LIN {X 0,Y 290.897,Z 639.692,A -85,B 0,C 180,E1 -29510.461,E2 -29510.461} C_VEL
LIN {X 0,Y 298.304,Z 601.913,A -85,B 0,C 180,E1 -29511.106,E2 -29511.106} C_VEL
LIN {X 0,Y 304.521,Z 561.656,A -85,B 0,C 180,E1 -29511.707,E2 -29511.707} C_VEL
LIN {X 0,Y 310.827,Z 508.179,A -85,B 0,C 180,E1 -29512.467,E2 -29512.467} C_VEL
LIN {X 0,Y 310.206,Z 504.294,A -85,B 0,C 180,E1 -29514.876,E2 -29514.876} C_VEL
LIN {X 0,Y 310.624,Z 502.045,A -85,B 0,C 180,E1 -29517.048,E2 -29517.048} C_VEL
LIN {X 0,Y 311.19,Z 500.451,A -85,B 0,C 180,E1 -29519.079,E2 -29519.079} C_VEL
LIN {X 0,Y 311.684,Z 500.279,A -85,B 0,C 180,E1 -29520.807,E2 -29520.807} C_VEL
LIN {X 0,Y 307.357,Z 520.155,A -85,B 0,C 180,E1 -29521.159,E2 -29521.159} C_VEL
LIN {X 0,Y 298.937,Z 587.892,A -85,B 0,C 180,E1 -29522.314,E2 -29522.314} C_VEL
LIN {X 0,Y 292.33,Z 627.482,A -85,B 0,C 180,E1 -29522.975,E2 -29522.975} C_VEL
LIN {X 0,Y 283.931,Z 667.082,A -85,B 0,C 180,E1 -29523.677,E2 -29523.677} C_VEL
LIN {X 0,Y 273.634,Z 706.852,A -85,B 0,C 180,E1 -29524.571,E2 -29524.571} C_VEL
LIN {X 0,Y 273.269,Z 708.115,A -85,B 0,C 180,E1 -29524.603,E2 -29524.603} C_VEL
LIN {X 0,Y 270.934,Z 715.53,A -85,B 0,C 180,E1 -29524.577,E2 -29524.577} C_VEL
LIN {X 0,Y 264.164,Z 735.315,A -85,B 0,C 180,E1 -29523.788,E2 -29523.788} C_VEL
LIN {X 0,Y 261.988,Z 741.59,A -85,B 0,C 180,E1 -29523.82,E2 -29523.82} C_VEL
LIN {X 0,Y 253.319,Z 766.281,A -85,B 0,C 180,E1 -29524.687,E2 -29524.687} C_VEL
LIN {X 0,Y 244.331,Z 786.818,A -85,B 0,C 180,E1 -29525.636,E2 -29525.636} C_VEL
LIN {X 0,Y 234.279,Z 805.781,A -85,B 0,C 180,E1 -29526.721,E2 -29526.721} C_VEL
LIN {X 0,Y 222.708,Z 824.293,A -85,B 0,C 180,E1 -29528.119,E2 -29528.119} C_VEL
LIN {X 0,Y 210.064,Z 841.669,A -85,B 0,C 180,E1 -29529.835,E2 -29529.835} C_VEL
LIN {X 0,Y 196.263,Z 858.133,A -85,B 0,C 180,E1 -29531.994,E2 -29531.994} C_VEL
LIN {X 0,Y 181.928,Z 873.186,A -85,B 0,C 180,E1 -29534.691,E2 -29534.691} C_VEL
LIN {X 0,Y 167.238,Z 886.889,A -85,B 0,C 180,E1 -29538.078,E2 -29538.078} C_VEL
LIN {X 0,Y 152.362,Z 899.309,A -85,B 0,C 180,E1 -29542.373,E2 -29542.373} C_VEL
LIN {X 0,Y 137.965,Z 910.277,A -85,B 0,C 180,E1 -29547.849,E2 -29547.849} C_VEL
LIN {X 0,Y 124.37,Z 919.877,A -85,B 0,C 180,E1 -29554.911,E2 -29554.911} C_VEL
LIN {X 0,Y 112.547,Z 927.982,A -85,B 0,C 180,E1 -29563.977,E2 -29563.977} C_VEL
LIN {X 0,Y 103.618,Z 934.442,A -85,B 0,C 180,E1 -29575.297,E2 -29575.297} C_VEL
LIN {X 0,Y 99.045,Z 938.841,A -85,B 0,C 180,E1 -29587.442,E2 -29587.442} C_VEL
LIN {X 0,Y 98.366,Z 941.455,A -85,B 0,C 180,E1 -29599.458,E2 -29599.458} C_VEL
LIN {X 0,Y 99.632,Z 942.357,A -85,B 0,C 180,E1 -29608.275,E2 -29608.275} C_VEL
LIN {X 0,Y 99.687,Z 942.359,A -85,B 0,C 180,E1 -29611.725,E2 -29611.725} C_VEL
LIN {X 0,Y 98.619,Z 941.398,A -85,B 0,C 180,E1 -29621.107,E2 -29621.107} C_VEL
LIN {X 0,Y 100.203,Z 938.422,A -85,B 0,C 180,E1 -29634.15,E2 -29634.15} C_VEL
LIN {X 0,Y 106.237,Z 933.564,A -85,B 0,C 180,E1 -29646.367,E2 -29646.367} C_VEL
LIN {X 0,Y 116.506,Z 926.832,A -85,B 0,C 180,E1 -29656.845,E2 -29656.845} C_VEL
LIN {X 0,Y 119.403,Z 925.309,A -85,B 0,C 180,E1 -29658.909,E2 -29658.909} C_VEL
LIN {X 0,Y 124.749,Z 925.094,A -85,B 0,C 180,E1 -29662.895,E2 -29662.895} C_VEL
LIN {X 0,Y 116.212,Z 919.228,A -85,B 0,C 180,E1 -29668.919,E2 -29668.919} C_VEL
LIN {X 0,Y 105.712,Z 915.062,A -85,B 0,C 180,E1 -29682.382,E2 -29682.382} C_VEL
LIN {X 0,Y 102.911,Z 908.863,A -85,B 0,C 180,E1 -29705.576,E2 -29705.576} C_VEL
LIN {X 0,Y 125.546,Z 900.271,A -85,B 0,C 180,E1 -29734.076,E2 -29734.076} C_VEL
LIN {X 0,Y 136.876,Z 897.562,A -85,B 0,C 180,E1 -29739.911,E2 -29739.911} C_VEL
LIN {X 0,Y 124.152,Z 904.891,A -85,B 0,C 180,E1 -29747.427,E2 -29747.427} C_VEL
LIN {X 0,Y 113.258,Z 910.617,A -85,B 0,C 180,E1 -29756.813,E2 -29756.813} C_VEL
LIN {X 0,Y 105.415,Z 914.504,A -85,B 0,C 180,E1 -29767.702,E2 -29767.702} C_VEL
LIN {X 0,Y 101.161,Z 916.605,A -85,B 0,C 180,E1 -29779.175,E2 -29779.175} C_VEL
LIN {X 0,Y 99.972,Z 917.237,A -85,B 0,C 180,E1 -29790.573,E2 -29790.573} C_VEL
LIN {X 0,Y 101.413,Z 916.524,A -85,B 0,C 180,E1 -29801.949,E2 -29801.949} C_VEL
LIN {X 0,Y 106.246,Z 914.18,A -85,B 0,C 180,E1 -29813.871,E2 -29813.871} C_VEL
LIN {X 0,Y 114.517,Z 910.086,A -85,B 0,C 180,E1 -29824.579,E2 -29824.579} C_VEL
LIN {X 0,Y 125.775,Z 904.102,A -85,B 0,C 180,E1 -29833.759,E2 -29833.759} C_VEL
LIN {X 0,Y 138.765,Z 896.517,A -85,B 0,C 180,E1 -29841.096,E2 -29841.096} C_VEL
LIN {X 0,Y 152.72,Z 887.421,A -85,B 0,C 180,E1 -29846.934,E2 -29846.934} C_VEL
LIN {X 0,Y 167.084,Z 876.867,A -85,B 0,C 180,E1 -29851.606,E2 -29851.606} C_VEL
LIN {X 0,Y 181.46,Z 864.89,A -85,B 0,C 180,E1 -29855.394,E2 -29855.394} C_VEL
LIN {X 0,Y 195.585,Z 851.485,A -85,B 0,C 180,E1 -29858.503,E2 -29858.503} C_VEL
LIN {X 0,Y 208.601,Z 837.38,A -85,B 0,C 180,E1 -29860.977,E2 -29860.977} C_VEL
LIN {X 0,Y 221.053,Z 821.901,A -85,B 0,C 180,E1 -29863.073,E2 -29863.073} C_VEL
LIN {X 0,Y 232.13,Z 806.011,A -85,B 0,C 180,E1 -29864.768,E2 -29864.768} C_VEL
LIN {X 0,Y 241.983,Z 789.593,A -85,B 0,C 180,E1 -29866.176,E2 -29866.176} C_VEL
LIN {X 0,Y 250.51,Z 772.939,A -85,B 0,C 180,E1 -29867.343,E2 -29867.343} C_VEL
LIN {X 0,Y 258.342,Z 754.518,A -85,B 0,C 180,E1 -29868.389,E2 -29868.389} C_VEL
LIN {X 0,Y 264.963,Z 735.092,A -85,B 0,C 180,E1 -29869.289,E2 -29869.289} C_VEL
LIN {X 0,Y 274.717,Z 701.51,A -85,B 0,C 180,E1 -29870.526,E2 -29870.526} C_VEL
LIN {X 0,Y 283.63,Z 667.686,A -85,B 0,C 180,E1 -29871.459,E2 -29871.459} C_VEL
LIN {X 0,Y 292.295,Z 629.172,A -85,B 0,C 180,E1 -29872.213,E2 -29872.213} C_VEL
LIN {X 0,Y 299.95,Z 586.992,A -85,B 0,C 180,E1 -29872.859,E2 -29872.859} C_VEL
LIN {X 0,Y 305.774,Z 544.445,A -85,B 0,C 180,E1 -29873.432,E2 -29873.432} C_VEL
LIN {X 0,Y 309.314,Z 514.061,A -85,B 0,C 180,E1 -29873.83,E2 -29873.83} C_VEL
LIN {X 0,Y 308.742,Z 510.419,A -85,B 0,C 180,E1 -29876.472,E2 -29876.472} C_VEL
LIN {X 0,Y 309.391,Z 508.21,A -85,B 0,C 180,E1 -29879.259,E2 -29879.259} C_VEL
LIN {X 0,Y 309.404,Z 508.336,A -85,B 0,C 180,E1 -29879.467,E2 -29879.467} C_VEL
LIN {X 0,Y 307.496,Z 517.679,A -85,B 0,C 180,E1 -29879.622,E2 -29879.622} C_VEL
LIN {X 0,Y 298.935,Z 585.198,A -85,B 0,C 180,E1 -29880.732,E2 -29880.732} C_VEL
LIN {X 0,Y 292.245,Z 624.865,A -85,B 0,C 180,E1 -29881.368,E2 -29881.368} C_VEL
LIN {X 0,Y 283.725,Z 664.756,A -85,B 0,C 180,E1 -29882.02,E2 -29882.02} C_VEL
LIN {X 0,Y 273.246,Z 704.978,A -85,B 0,C 180,E1 -29882.855,E2 -29882.855} C_VEL
LIN {X 0,Y 261.988,Z 741.59,A -85,B 0,C 180,E1 -29883.82,E2 -29883.82} C_VEL
LIN {X 0,Y 259.38,Z 748.91,A -85,B 0,C 180,E1 -29883.841,E2 -29883.841} C_VEL
LIN {X 0,Y 252.021,Z 767.378,A -85,B 0,C 180,E1 -29883.147,E2 -29883.147} C_VEL
LIN {X 0,Y 248.861,Z 774.441,A -85,B 0,C 180,E1 -29883.206,E2 -29883.206} C_VEL
LIN {X 0,Y 239.587,Z 793.606,A -85,B 0,C 180,E1 -29884.102,E2 -29884.102} C_VEL
LIN {X 0,Y 228.912,Z 812.088,A -85,B 0,C 180,E1 -29885.187,E2 -29885.187} C_VEL
LIN {X 0,Y 216.891,Z 829.847,A -85,B 0,C 180,E1 -29886.549,E2 -29886.549} C_VEL
LIN {X 0,Y 203.66,Z 846.745,A -85,B 0,C 180,E1 -29888.28,E2 -29888.28} C_VEL
LIN {X 0,Y 189.138,Z 862.871,A -85,B 0,C 180,E1 -29890.487,E2 -29890.487} C_VEL
LIN {X 0,Y 173.667,Z 877.908,A -85,B 0,C 180,E1 -29893.34,E2 -29893.34} C_VEL
LIN {X 0,Y 157.883,Z 891.47,A -85,B 0,C 180,E1 -29897.001,E2 -29897.001} C_VEL
LIN {X 0,Y 142.882,Z 902.971,A -85,B 0,C 180,E1 -29901.451,E2 -29901.451} C_VEL
LIN {X 0,Y 128.217,Z 913.193,A -85,B 0,C 180,E1 -29907.25,E2 -29907.25} C_VEL
LIN {X 0,Y 114.514,Z 922.062,A -85,B 0,C 180,E1 -29914.839,E2 -29914.839} C_VEL
LIN {X 0,Y 102.767,Z 929.47,A -85,B 0,C 180,E1 -29924.744,E2 -29924.744} C_VEL
LIN {X 0,Y 94.278,Z 935.285,A -85,B 0,C 180,E1 -29937.256,E2 -29937.256} C_VEL
LIN {X 0,Y 90.532,Z 939.048,A -85,B 0,C 180,E1 -29950.651,E2 -29950.651} C_VEL
LIN {X 0,Y 90.763,Z 940.997,A -85,B 0,C 180,E1 -29963.04,E2 -29963.04} C_VEL
LIN {X 0,Y 91.884,Z 941.432,A -85,B 0,C 180,E1 -29970,E2 -29970} C_VEL
LIN {X 0,Y 90.836,Z 940.851,A -85,B 0,C 180,E1 -29978.228,E2 -29978.228} C_VEL
LIN {X 0,Y 91.414,Z 938.653,A -85,B 0,C 180,E1 -29991.159,E2 -29991.159} C_VEL
LIN {X 0,Y 96.614,Z 934.465,A -85,B 0,C 180,E1 -30004.696,E2 -30004.696} C_VEL
LIN {X 0,Y 106.466,Z 928.428,A -85,B 0,C 180,E1 -30016.317,E2 -30016.317} C_VEL
LIN {X 0,Y 115.043,Z 923.428,A -85,B 0,C 180,E1 -30022.69,E2 -30022.69} C_VEL
LIN {X 0,Y 98.283,Z 917.708,A -85,B 0,C 180,E1 -30041.616,E2 -30041.616} C_VEL
LIN {X 0,Y 95.574,Z 911.594,A -85,B 0,C 180,E1 -30066.608,E2 -30066.608} C_VEL
LIN {X 0,Y 120.481,Z 902.974,A -85,B 0,C 180,E1 -30096.694,E2 -30096.694} C_VEL
LIN {X 0,Y 126.523,Z 901.616,A -85,B 0,C 180,E1 -30099.952,E2 -30099.952} C_VEL
LIN {X 0,Y 113.258,Z 908.513,A -85,B 0,C 180,E1 -30108.537,E2 -30108.537} C_VEL
LIN {X 0,Y 102.737,Z 913.467,A -85,B 0,C 180,E1 -30118.947,E2 -30118.947} C_VEL
LIN {X 0,Y 95.637,Z 916.618,A -85,B 0,C 180,E1 -30131.088,E2 -30131.088} C_VEL
LIN {X 0,Y 92.398,Z 918.07,A -85,B 0,C 180,E1 -30143.787,E2 -30143.787} C_VEL
LIN {X 0,Y 92.317,Z 918.094,A -85,B 0,C 180,E1 -30155.594,E2 -30155.594} C_VEL
LIN {X 0,Y 95.148,Z 916.84,A -85,B 0,C 180,E1 -30167.743,E2 -30167.743} C_VEL
LIN {X 0,Y 101.501,Z 914.044,A -85,B 0,C 180,E1 -30179.508,E2 -30179.508} C_VEL
LIN {X 0,Y 111.054,Z 909.628,A -85,B 0,C 180,E1 -30189.736,E2 -30189.736} C_VEL
LIN {X 0,Y 123.245,Z 903.471,A -85,B 0,C 180,E1 -30198.297,E2 -30198.297} C_VEL
LIN {X 0,Y 136.712,Z 895.88,A -85,B 0,C 180,E1 -30205,E2 -30205} C_VEL
LIN {X 0,Y 150.811,Z 886.928,A -85,B 0,C 180,E1 -30210.289,E2 -30210.289} C_VEL
LIN {X 0,Y 165.299,Z 876.511,A -85,B 0,C 180,E1 -30214.565,E2 -30214.565} C_VEL
LIN {X 0,Y 179.131,Z 865.234,A -85,B 0,C 180,E1 -30217.909,E2 -30217.909} C_VEL
LIN {X 0,Y 192.812,Z 852.576,A -85,B 0,C 180,E1 -30220.703,E2 -30220.703} C_VEL
LIN {X 0,Y 205.944,Z 838.715,A -85,B 0,C 180,E1 -30223.031,E2 -30223.031} C_VEL
LIN {X 0,Y 218.425,Z 823.602,A -85,B 0,C 180,E1 -30224.994,E2 -30224.994} C_VEL
LIN {X 0,Y 229.719,Z 807.819,A -85,B 0,C 180,E1 -30226.611,E2 -30226.611} C_VEL
LIN {X 0,Y 239.896,Z 791.267,A -85,B 0,C 180,E1 -30227.971,E2 -30227.971} C_VEL
LIN {X 0,Y 248.796,Z 774.223,A -85,B 0,C 180,E1 -30229.112,E2 -30229.112} C_VEL
LIN {X 0,Y 256.326,Z 757.022,A -85,B 0,C 180,E1 -30230.052,E2 -30230.052} C_VEL
LIN {X 0,Y 263.199,Z 737.453,A -85,B 0,C 180,E1 -30230.931,E2 -30230.931} C_VEL
LIN {X 0,Y 273.439,Z 703.168,A -85,B 0,C 180,E1 -30232.149,E2 -30232.149} C_VEL
LIN {X 0,Y 282.636,Z 668.648,A -85,B 0,C 180,E1 -30233.055,E2 -30233.055} C_VEL
LIN {X 0,Y 291.108,Z 631.644,A -85,B 0,C 180,E1 -30233.744,E2 -30233.744} C_VEL
LIN {X 0,Y 298.841,Z 589.7,A -85,B 0,C 180,E1 -30234.349,E2 -30234.349} C_VEL
LIN {X 0,Y 304.708,Z 547.493,A -85,B 0,C 180,E1 -30234.891,E2 -30234.891} C_VEL
LIN {X 0,Y 307.943,Z 520.078,A -85,B 0,C 180,E1 -30235.251,E2 -30235.251} C_VEL
LIN {X 0,Y 307.644,Z 517.482,A -85,B 0,C 180,E1 -30237.578,E2 -30237.578} C_VEL
LIN {X 0,Y 307.613,Z 517.161,A -85,B 0,C 180,E1 -30238.118,E2 -30238.118} C_VEL
LIN {X 0,Y 299.156,Z 582.532,A -85,B 0,C 180,E1 -30239.151,E2 -30239.151} C_VEL
LIN {X 0,Y 292.354,Z 622.416,A -85,B 0,C 180,E1 -30239.765,E2 -30239.765} C_VEL
LIN {X 0,Y 283.768,Z 662.379,A -85,B 0,C 180,E1 -30240.361,E2 -30240.361} C_VEL
LIN {X 0,Y 273.179,Z 702.835,A -85,B 0,C 180,E1 -30241.131,E2 -30241.131} C_VEL
LIN {X 0,Y 261.634,Z 740.122,A -85,B 0,C 180,E1 -30242.025,E2 -30242.025} C_VEL
LIN {X 0,Y 252.78,Z 765.045,A -85,B 0,C 180,E1 -30242.831,E2 -30242.831} C_VEL
LIN {X 0,Y 248.861,Z 774.441,A -85,B 0,C 180,E1 -30243.206,E2 -30243.206} C_VEL
LIN {X 0,Y 245.416,Z 781.76,A -85,B 0,C 180,E1 -30243.289,E2 -30243.289} C_VEL
LIN {X 0,Y 235.59,Z 799.083,A -85,B 0,C 180,E1 -30242.693,E2 -30242.693} C_VEL
LIN {X 0,Y 231.635,Z 805.444,A -85,B 0,C 180,E1 -30242.799,E2 -30242.799} C_VEL
LIN {X 0,Y 220.49,Z 822.504,A -85,B 0,C 180,E1 -30243.914,E2 -30243.914} C_VEL
LIN {X 0,Y 208.44,Z 838.497,A -85,B 0,C 180,E1 -30245.229,E2 -30245.229} C_VEL
LIN {X 0,Y 194.433,Z 854.698,A -85,B 0,C 180,E1 -30247.014,E2 -30247.014} C_VEL
LIN {X 0,Y 179.35,Z 869.944,A -85,B 0,C 180,E1 -30249.324,E2 -30249.324} C_VEL
LIN {X 0,Y 163.704,Z 883.811,A -85,B 0,C 180,E1 -30252.241,E2 -30252.241} C_VEL
LIN {X 0,Y 147.139,Z 896.754,A -85,B 0,C 180,E1 -30256.178,E2 -30256.178} C_VEL
LIN {X 0,Y 130.928,Z 908.015,A -85,B 0,C 180,E1 -30261.298,E2 -30261.298} C_VEL
LIN {X 0,Y 115.543,Z 917.657,A -85,B 0,C 180,E1 -30268.032,E2 -30268.032} C_VEL
LIN {X 0,Y 101.578,Z 925.785,A -85,B 0,C 180,E1 -30277.125,E2 -30277.125} C_VEL
LIN {X 0,Y 90.768,Z 932.047,A -85,B 0,C 180,E1 -30288.628,E2 -30288.628} C_VEL
LIN {X 0,Y 84.153,Z 936.564,A -85,B 0,C 180,E1 -30302.394,E2 -30302.394} C_VEL
LIN {X 0,Y 82.324,Z 939.385,A -85,B 0,C 180,E1 -30317.372,E2 -30317.372} C_VEL
LIN {X 0,Y 83.705,Z 940.369,A -85,B 0,C 180,E1 -30328.631,E2 -30328.631} C_VEL
LIN {X 0,Y 83.795,Z 940.376,A -85,B 0,C 180,E1 -30331.368,E2 -30331.368} C_VEL
LIN {X 0,Y 82.683,Z 939.337,A -85,B 0,C 180,E1 -30343.284,E2 -30343.284} C_VEL
LIN {X 0,Y 85.426,Z 936.323,A -85,B 0,C 180,E1 -30358.679,E2 -30358.679} C_VEL
LIN {X 0,Y 93.941,Z 931.168,A -85,B 0,C 180,E1 -30372.939,E2 -30372.939} C_VEL
LIN {X 0,Y 105.206,Z 924.983,A -85,B 0,C 180,E1 -30383.049,E2 -30383.049} C_VEL
LIN {X 0,Y 87.962,Z 914.352,A -85,B 0,C 180,E1 -30426.527,E2 -30426.527} C_VEL
LIN {X 0,Y 113.972,Z 905.824,A -85,B 0,C 180,E1 -30458.665,E2 -30458.665} C_VEL
LIN {X 0,Y 116.137,Z 905.376,A -85,B 0,C 180,E1 -30459.981,E2 -30459.981} C_VEL
LIN {X 0,Y 102.89,Z 911.534,A -85,B 0,C 180,E1 -30469.374,E2 -30469.374} C_VEL
LIN {X 0,Y 92.681,Z 915.818,A -85,B 0,C 180,E1 -30480.956,E2 -30480.956} C_VEL
LIN {X 0,Y 86.506,Z 918.256,A -85,B 0,C 180,E1 -30493.894,E2 -30493.894} C_VEL
LIN {X 0,Y 84.155,Z 919.174,A -85,B 0,C 180,E1 -30507.275,E2 -30507.275} C_VEL
LIN {X 0,Y 85.139,Z 918.795,A -85,B 0,C 180,E1 -30520.83,E2 -30520.83} C_VEL
LIN {X 0,Y 89.844,Z 916.965,A -85,B 0,C 180,E1 -30534.316,E2 -30534.316} C_VEL
LIN {X 0,Y 98.736,Z 913.368,A -85,B 0,C 180,E1 -30546.69,E2 -30546.69} C_VEL
LIN {X 0,Y 110.955,Z 907.949,A -85,B 0,C 180,E1 -30556.881,E2 -30556.881} C_VEL
LIN {X 0,Y 124.281,Z 901.313,A -85,B 0,C 180,E1 -30564.349,E2 -30564.349} C_VEL
LIN {X 0,Y 138.369,Z 893.378,A -85,B 0,C 180,E1 -30570.128,E2 -30570.128} C_VEL
LIN {X 0,Y 153.498,Z 883.669,A -85,B 0,C 180,E1 -30574.883,E2 -30574.883} C_VEL
LIN {X 0,Y 168.553,Z 872.614,A -85,B 0,C 180,E1 -30578.647,E2 -30578.647} C_VEL
LIN {X 0,Y 183.271,Z 860.256,A -85,B 0,C 180,E1 -30581.679,E2 -30581.679} C_VEL
LIN {X 0,Y 197.009,Z 847.042,A -85,B 0,C 180,E1 -30584.093,E2 -30584.093} C_VEL
LIN {X 0,Y 210.573,Z 832.06,A -85,B 0,C 180,E1 -30586.18,E2 -30586.18} C_VEL
LIN {X 0,Y 222.939,Z 816.241,A -85,B 0,C 180,E1 -30587.887,E2 -30587.887} C_VEL
LIN {X 0,Y 234.043,Z 799.685,A -85,B 0,C 180,E1 -30589.302,E2 -30589.302} C_VEL
LIN {X 0,Y 244.295,Z 781.633,A -85,B 0,C 180,E1 -30590.541,E2 -30590.541} C_VEL
LIN {X 0,Y 252.728,Z 763.766,A -85,B 0,C 180,E1 -30591.531,E2 -30591.531} C_VEL
LIN {X 0,Y 260.245,Z 744.124,A -85,B 0,C 180,E1 -30592.421,E2 -30592.421} C_VEL
LIN {X 0,Y 270.885,Z 710.049,A -85,B 0,C 180,E1 -30593.627,E2 -30593.627} C_VEL
LIN {X 0,Y 280.975,Z 673.445,A -85,B 0,C 180,E1 -30594.581,E2 -30594.581} C_VEL
LIN {X 0,Y 289.674,Z 636.145,A -85,B 0,C 180,E1 -30595.255,E2 -30595.255} C_VEL
LIN {X 0,Y 297.291,Z 596.18,A -85,B 0,C 180,E1 -30595.8,E2 -30595.8} C_VEL
LIN {X 0,Y 303.116,Z 556.268,A -85,B 0,C 180,E1 -30596.293,E2 -30596.293} C_VEL
LIN {X 0,Y 306.729,Z 526.374,A -85,B 0,C 180,E1 -30596.683,E2 -30596.683} C_VEL
LIN {X 0,Y 306.69,Z 526.528,A -85,B 0,C 180,E1 -30596.765,E2 -30596.765} C_VEL
LIN {X 0,Y 299.179,Z 582.552,A -85,B 0,C 180,E1 -30597.615,E2 -30597.615} C_VEL
LIN {X 0,Y 292.333,Z 621.691,A -85,B 0,C 180,E1 -30598.186,E2 -30598.186} C_VEL
LIN {X 0,Y 283.917,Z 660.513,A -85,B 0,C 180,E1 -30598.713,E2 -30598.713} C_VEL
LIN {X 0,Y 273.328,Z 700.792,A -85,B 0,C 180,E1 -30599.409,E2 -30599.409} C_VEL
LIN {X 0,Y 261.972,Z 737.428,A -85,B 0,C 180,E1 -30600.198,E2 -30600.198} C_VEL
LIN {X 0,Y 253.005,Z 762.644,A -85,B 0,C 180,E1 -30600.929,E2 -30600.929} C_VEL
LIN {X 0,Y 244.576,Z 781.78,A -85,B 0,C 180,E1 -30601.659,E2 -30601.659} C_VEL
LIN {X 0,Y 234.209,Z 801.18,A -85,B 0,C 180,E1 -30602.567,E2 -30602.567} C_VEL
LIN {X 0,Y 231.635,Z 805.444,A -85,B 0,C 180,E1 -30602.799,E2 -30602.799} C_VEL
LIN {X 0,Y 227.51,Z 812.018,A -85,B 0,C 180,E1 -30602.93,E2 -30602.93} C_VEL
LIN {X 0,Y 215.454,Z 828.05,A -85,B 0,C 180,E1 -30602.458,E2 -30602.458} C_VEL
LIN {X 0,Y 210.544,Z 834.011,A -85,B 0,C 180,E1 -30602.661,E2 -30602.661} C_VEL
LIN {X 0,Y 196.509,Z 850.413,A -85,B 0,C 180,E1 -30604.213,E2 -30604.213} C_VEL
LIN {X 0,Y 182.009,Z 865.202,A -85,B 0,C 180,E1 -30606.097,E2 -30606.097} C_VEL
LIN {X 0,Y 165.684,Z 879.722,A -85,B 0,C 180,E1 -30608.678,E2 -30608.678} C_VEL
LIN {X 0,Y 149.238,Z 892.561,A -85,B 0,C 180,E1 -30611.988,E2 -30611.988} C_VEL
LIN {X 0,Y 132.381,Z 904.133,A -85,B 0,C 180,E1 -30616.415,E2 -30616.415} C_VEL
LIN {X 0,Y 114.956,Z 914.714,A -85,B 0,C 180,E1 -30622.781,E2 -30622.781} C_VEL
LIN {X 0,Y 99.405,Z 923.251,A -85,B 0,C 180,E1 -30631.242,E2 -30631.242} C_VEL
LIN {X 0,Y 86.671,Z 929.904,A -85,B 0,C 180,E1 -30642.41,E2 -30642.41} C_VEL
LIN {X 0,Y 77.683,Z 934.991,A -85,B 0,C 180,E1 -30657.276,E2 -30657.276} C_VEL
LIN {X 0,Y 74.38,Z 938.082,A -85,B 0,C 180,E1 -30673.603,E2 -30673.603} C_VEL
LIN {X 0,Y 75.401,Z 939.275,A -85,B 0,C 180,E1 -30686.96,E2 -30686.96} C_VEL
LIN {X 0,Y 75.898,Z 939.4,A -85,B 0,C 180,E1 -30690.755,E2 -30690.755} C_VEL
LIN {X 0,Y 74.73,Z 938.387,A -85,B 0,C 180,E1 -30703.937,E2 -30703.937} C_VEL
LIN {X 0,Y 78.008,Z 935.438,A -85,B 0,C 180,E1 -30720.845,E2 -30720.845} C_VEL
LIN {X 0,Y 87.07,Z 930.614,A -85,B 0,C 180,E1 -30735.532,E2 -30735.532} C_VEL
LIN {X 0,Y 95.561,Z 926.36,A -85,B 0,C 180,E1 -30743.387,E2 -30743.387} C_VEL
LIN {X 0,Y 80.507,Z 916.643,A -85,B 0,C 180,E1 -30787.852,E2 -30787.852} C_VEL
LIN {X 0,Y 105.806,Z 908.837,A -85,B 0,C 180,E1 -30819.941,E2 -30819.941} C_VEL
LIN {X 0,Y 92.509,Z 914.309,A -85,B 0,C 180,E1 -30830.378,E2 -30830.378} C_VEL
LIN {X 0,Y 82.543,Z 917.978,A -85,B 0,C 180,E1 -30843.69,E2 -30843.69} C_VEL
LIN {X 0,Y 77.216,Z 919.83,A -85,B 0,C 180,E1 -30858.799,E2 -30858.799} C_VEL
LIN {X 0,Y 76.265,Z 920.164,A -85,B 0,C 180,E1 -30873.758,E2 -30873.758} C_VEL
LIN {X 0,Y 79.269,Z 919.146,A -85,B 0,C 180,E1 -30888.906,E2 -30888.906} C_VEL
LIN {X 0,Y 86.613,Z 916.566,A -85,B 0,C 180,E1 -30902.859,E2 -30902.859} C_VEL
LIN {X 0,Y 97.498,Z 912.41,A -85,B 0,C 180,E1 -30914.216,E2 -30914.216} C_VEL
LIN {X 0,Y 111.108,Z 906.536,A -85,B 0,C 180,E1 -30923.219,E2 -30923.219} C_VEL
LIN {X 0,Y 125.894,Z 899.224,A -85,B 0,C 180,E1 -30929.975,E2 -30929.975} C_VEL
LIN {X 0,Y 141.089,Z 890.591,A -85,B 0,C 180,E1 -30935.111,E2 -30935.111} C_VEL
LIN {X 0,Y 156.263,Z 880.695,A -85,B 0,C 180,E1 -30939.101,E2 -30939.101} C_VEL
LIN {X 0,Y 171.564,Z 869.227,A -85,B 0,C 180,E1 -30942.358,E2 -30942.358} C_VEL
LIN {X 0,Y 185.439,Z 857.363,A -85,B 0,C 180,E1 -30944.833,E2 -30944.833} C_VEL
LIN {X 0,Y 199.581,Z 843.46,A -85,B 0,C 180,E1 -30947.016,E2 -30947.016} C_VEL
LIN {X 0,Y 212.537,Z 828.799,A -85,B 0,C 180,E1 -30948.783,E2 -30948.783} C_VEL
LIN {X 0,Y 224.695,Z 812.848,A -85,B 0,C 180,E1 -30950.289,E2 -30950.289} C_VEL
LIN {X 0,Y 235.537,Z 796.244,A -85,B 0,C 180,E1 -30951.54,E2 -30951.54} C_VEL
LIN {X 0,Y 245.494,Z 778.148,A -85,B 0,C 180,E1 -30952.643,E2 -30952.643} C_VEL
LIN {X 0,Y 254.068,Z 759.222,A -85,B 0,C 180,E1 -30953.574,E2 -30953.574} C_VEL
LIN {X 0,Y 261.948,Z 737.318,A -85,B 0,C 180,E1 -30954.451,E2 -30954.451} C_VEL
LIN {X 0,Y 272.925,Z 701.674,A -85,B 0,C 180,E1 -30955.564,E2 -30955.564} C_VEL
LIN {X 0,Y 282.567,Z 665.722,A -85,B 0,C 180,E1 -30956.368,E2 -30956.368} C_VEL
LIN {X 0,Y 288.838,Z 638.838,A -85,B 0,C 180,E1 -30956.812,E2 -30956.812} C_VEL
LIN {X 0,Y 279.381,Z 678.226,A -85,B 0,C 180,E1 -30957.357,E2 -30957.357} C_VEL
LIN {X 0,Y 267.773,Z 718.617,A -85,B 0,C 180,E1 -30958.05,E2 -30958.05} C_VEL
LIN {X 0,Y 256.526,Z 752.173,A -85,B 0,C 180,E1 -30958.819,E2 -30958.819} C_VEL
LIN {X 0,Y 248.987,Z 770.899,A -85,B 0,C 180,E1 -30959.378,E2 -30959.378} C_VEL
LIN {X 0,Y 239.61,Z 789.996,A -85,B 0,C 180,E1 -30960.109,E2 -30960.109} C_VEL
LIN {X 0,Y 229.006,Z 808.108,A -85,B 0,C 180,E1 -30960.956,E2 -30960.956} C_VEL
LIN {X 0,Y 216.618,Z 826.107,A -85,B 0,C 180,E1 -30962.078,E2 -30962.078} C_VEL
LIN {X 0,Y 210.544,Z 834.011,A -85,B 0,C 180,E1 -30962.661,E2 -30962.661} C_VEL
LIN {X 0,Y 205.457,Z 840.042,A -85,B 0,C 180,E1 -30962.896,E2 -30962.896} C_VEL
LIN {X 0,Y 191.375,Z 854.341,A -85,B 0,C 180,E1 -30962.589,E2 -30962.589} C_VEL
LIN {X 0,Y 185.894,Z 859.552,A -85,B 0,C 180,E1 -30962.898,E2 -30962.898} C_VEL
LIN {X 0,Y 170.604,Z 873.527,A -85,B 0,C 180,E1 -30964.9,E2 -30964.9} C_VEL
LIN {X 0,Y 154.315,Z 886.567,A -85,B 0,C 180,E1 -30967.533,E2 -30967.533} C_VEL
LIN {X 0,Y 137.515,Z 898.345,A -85,B 0,C 180,E1 -30971.008,E2 -30971.008} C_VEL
LIN {X 0,Y 119.64,Z 909.329,A -85,B 0,C 180,E1 -30976.032,E2 -30976.032} C_VEL
LIN {X 0,Y 102.455,Z 918.607,A -85,B 0,C 180,E1 -30982.978,E2 -30982.978} C_VEL
LIN {X 0,Y 86.876,Z 926.217,A -85,B 0,C 180,E1 -30992.841,E2 -30992.841} C_VEL
LIN {X 0,Y 74.43,Z 932.075,A -85,B 0,C 180,E1 -31006.754,E2 -31006.754} C_VEL
LIN {X 0,Y 67.439,Z 936.029,A -85,B 0,C 180,E1 -31024.535,E2 -31024.535} C_VEL
LIN {X 0,Y 66.746,Z 938.029,A -85,B 0,C 180,E1 -31042.252,E2 -31042.252} C_VEL
LIN {X 0,Y 67.871,Z 938.388,A -85,B 0,C 180,E1 -31050.845,E2 -31050.845} C_VEL
LIN {X 0,Y 66.823,Z 937.354,A -85,B 0,C 180,E1 -31065.626,E2 -31065.626} C_VEL
LIN {X 0,Y 71.035,Z 934.386,A -85,B 0,C 180,E1 -31084.267,E2 -31084.267} C_VEL
LIN {X 0,Y 81.389,Z 929.589,A -85,B 0,C 180,E1 -31099.614,E2 -31099.614} C_VEL
LIN {X 0,Y 85.695,Z 927.592,A -85,B 0,C 180,E1 -31103.745,E2 -31103.745} C_VEL
LIN {X 0,Y 73.049,Z 918.736,A -85,B 0,C 180,E1 -31149.454,E2 -31149.454} C_VEL
LIN {X 0,Y 95.351,Z 912.093,A -85,B 0,C 180,E1 -31179.932,E2 -31179.932} C_VEL
LIN {X 0,Y 82.095,Z 916.861,A -85,B 0,C 180,E1 -31191.598,E2 -31191.598} C_VEL
LIN {X 0,Y 72.797,Z 919.826,A -85,B 0,C 180,E1 -31206.526,E2 -31206.526} C_VEL
LIN {X 0,Y 68.659,Z 921.092,A -85,B 0,C 180,E1 -31222.468,E2 -31222.468} C_VEL
LIN {X 0,Y 68.75,Z 921.084,A -85,B 0,C 180,E1 -31238.362,E2 -31238.362} C_VEL
LIN {X 0,Y 73.417,Z 919.686,A -85,B 0,C 180,E1 -31254.973,E2 -31254.973} C_VEL
LIN {X 0,Y 83.239,Z 916.568,A -85,B 0,C 180,E1 -31269.754,E2 -31269.754} C_VEL
LIN {X 0,Y 96.56,Z 911.731,A -85,B 0,C 180,E1 -31280.953,E2 -31280.953} C_VEL
LIN {X 0,Y 111.815,Z 905.264,A -85,B 0,C 180,E1 -31289.144,E2 -31289.144} C_VEL
LIN {X 0,Y 127.821,Z 897.347,A -85,B 0,C 180,E1 -31295.15,E2 -31295.15} C_VEL
LIN {X 0,Y 144.067,Z 887.991,A -85,B 0,C 180,E1 -31299.695,E2 -31299.695} C_VEL
LIN {X 0,Y 159.837,Z 877.473,A -85,B 0,C 180,E1 -31303.16,E2 -31303.16} C_VEL
LIN {X 0,Y 175.24,Z 865.614,A -85,B 0,C 180,E1 -31305.928,E2 -31305.928} C_VEL
LIN {X 0,Y 190.012,Z 852.493,A -85,B 0,C 180,E1 -31308.174,E2 -31308.174} C_VEL
LIN {X 0,Y 204.526,Z 837.542,A -85,B 0,C 180,E1 -31310.095,E2 -31310.095} C_VEL
LIN {X 0,Y 217.737,Z 821.729,A -85,B 0,C 180,E1 -31311.654,E2 -31311.654} C_VEL
LIN {X 0,Y 229.709,Z 804.958,A -85,B 0,C 180,E1 -31312.954,E2 -31312.954} C_VEL
LIN {X 0,Y 240.953,Z 786.217,A -85,B 0,C 180,E1 -31314.114,E2 -31314.114} C_VEL
LIN {X 0,Y 249.917,Z 768.175,A -85,B 0,C 180,E1 -31315.016,E2 -31315.016} C_VEL
LIN {X 0,Y 257.662,Z 748.98,A -85,B 0,C 180,E1 -31315.805,E2 -31315.805} C_VEL
LIN {X 0,Y 264.634,Z 728.339,A -85,B 0,C 180,E1 -31316.513,E2 -31316.513} C_VEL
LIN {X 0,Y 254.792,Z 756.595,A -85,B 0,C 180,E1 -31317.128,E2 -31317.128} C_VEL
LIN {X 0,Y 245.665,Z 777.367,A -85,B 0,C 180,E1 -31317.733,E2 -31317.733} C_VEL
LIN {X 0,Y 235.058,Z 797.078,A -85,B 0,C 180,E1 -31318.463,E2 -31318.463} C_VEL
LIN {X 0,Y 223.491,Z 815.191,A -85,B 0,C 180,E1 -31319.311,E2 -31319.311} C_VEL
LIN {X 0,Y 210.689,Z 832.347,A -85,B 0,C 180,E1 -31320.367,E2 -31320.367} C_VEL
LIN {X 0,Y 196.409,Z 848.853,A -85,B 0,C 180,E1 -31321.75,E2 -31321.75} C_VEL
LIN {X 0,Y 185.894,Z 859.552,A -85,B 0,C 180,E1 -31322.898,E2 -31322.898} C_VEL
LIN {X 0,Y 180.234,Z 864.781,A -85,B 0,C 180,E1 -31323.251,E2 -31323.251} C_VEL
LIN {X 0,Y 164.422,Z 877.237,A -85,B 0,C 180,E1 -31323.174,E2 -31323.174} C_VEL
LIN {X 0,Y 158.338,Z 881.828,A -85,B 0,C 180,E1 -31323.662,E2 -31323.662} C_VEL
LIN {X 0,Y 139.96,Z 894.787,A -85,B 0,C 180,E1 -31326.769,E2 -31326.769} C_VEL
LIN {X 0,Y 121.877,Z 905.816,A -85,B 0,C 180,E1 -31330.877,E2 -31330.877} C_VEL
LIN {X 0,Y 104.292,Z 915.147,A -85,B 0,C 180,E1 -31336.516,E2 -31336.516} C_VEL
LIN {X 0,Y 87.099,Z 923.149,A -85,B 0,C 180,E1 -31344.918,E2 -31344.918} C_VEL
LIN {X 0,Y 71.823,Z 929.609,A -85,B 0,C 180,E1 -31357.774,E2 -31357.774} C_VEL
LIN {X 0,Y 61.693,Z 934.058,A -85,B 0,C 180,E1 -31375.441,E2 -31375.441} C_VEL
LIN {X 0,Y 58.442,Z 936.624,A -85,B 0,C 180,E1 -31396.142,E2 -31396.142} C_VEL
LIN {X 0,Y 59.907,Z 937.393,A -85,B 0,C 180,E1 -31410.479,E2 -31410.479} C_VEL
LIN {X 0,Y 59.056,Z 936.255,A -85,B 0,C 180,E1 -31428.532,E2 -31428.532} C_VEL
LIN {X 0,Y 64.789,Z 933.168,A -85,B 0,C 180,E1 -31449.254,E2 -31449.254} C_VEL
LIN {X 0,Y 76.025,Z 928.598,A -85,B 0,C 180,E1 -31464.21,E2 -31464.21} C_VEL
LIN {X 0,Y 65.603,Z 920.585,A -85,B 0,C 180,E1 -31511.428,E2 -31511.428} C_VEL
LIN {X 0,Y 84.945,Z 915.027,A -85,B 0,C 180,E1 -31539.819,E2 -31539.819} C_VEL
LIN {X 0,Y 71.674,Z 919.179,A -85,B 0,C 180,E1 -31553.138,E2 -31553.138} C_VEL
LIN {X 0,Y 63.076,Z 921.525,A -85,B 0,C 180,E1 -31570.555,E2 -31570.555} C_VEL
LIN {X 0,Y 60.291,Z 922.231,A -85,B 0,C 180,E1 -31589.049,E2 -31589.049} C_VEL
LIN {X 0,Y 62.548,Z 921.649,A -85,B 0,C 180,E1 -31607.681,E2 -31607.681} C_VEL
LIN {X 0,Y 70.154,Z 919.62,A -85,B 0,C 180,E1 -31624.758,E2 -31624.758} C_VEL
LIN {X 0,Y 82.083,Z 916.03,A -85,B 0,C 180,E1 -31637.993,E2 -31637.993} C_VEL
LIN {X 0,Y 96.938,Z 910.777,A -85,B 0,C 180,E1 -31647.758,E2 -31647.758} C_VEL
LIN {X 0,Y 113.675,Z 903.742,A -85,B 0,C 180,E1 -31654.957,E2 -31654.957} C_VEL
LIN {X 0,Y 131.632,Z 894.76,A -85,B 0,C 180,E1 -31660.376,E2 -31660.376} C_VEL
LIN {X 0,Y 148.59,Z 884.696,A -85,B 0,C 180,E1 -31664.211,E2 -31664.211} C_VEL
LIN {X 0,Y 165.096,Z 873.242,A -85,B 0,C 180,E1 -31667.181,E2 -31667.181} C_VEL
LIN {X 0,Y 180.985,Z 860.422,A -85,B 0,C 180,E1 -31669.544,E2 -31669.544} C_VEL
LIN {X 0,Y 196.146,Z 846.214,A -85,B 0,C 180,E1 -31671.474,E2 -31671.474} C_VEL
LIN {X 0,Y 210.508,Z 830.508,A -85,B 0,C 180,E1 -31673.084,E2 -31673.084} C_VEL
LIN {X 0,Y 224.023,Z 813.118,A -85,B 0,C 180,E1 -31674.457,E2 -31674.457} C_VEL
LIN {X 0,Y 235.191,Z 796.122,A -85,B 0,C 180,E1 -31675.523,E2 -31675.523} C_VEL
LIN {X 0,Y 241.418,Z 785.307,A -85,B 0,C 180,E1 -31676.101,E2 -31676.101} C_VEL
LIN {X 0,Y 230.336,Z 804.144,A -85,B 0,C 180,E1 -31676.765,E2 -31676.765} C_VEL
LIN {X 0,Y 218.169,Z 821.724,A -85,B 0,C 180,E1 -31677.585,E2 -31677.585} C_VEL
LIN {X 0,Y 204.596,Z 838.546,A -85,B 0,C 180,E1 -31678.6,E2 -31678.6} C_VEL
LIN {X 0,Y 189.479,Z 854.705,A -85,B 0,C 180,E1 -31679.948,E2 -31679.948} C_VEL
LIN {X 0,Y 173.747,Z 869.308,A -85,B 0,C 180,E1 -31681.649,E2 -31681.649} C_VEL
LIN {X 0,Y 158.338,Z 881.828,A -85,B 0,C 180,E1 -31683.662,E2 -31683.662} C_VEL
LIN {X 0,Y 152.133,Z 886.259,A -85,B 0,C 180,E1 -31684.213,E2 -31684.213} C_VEL
LIN {X 0,Y 134.855,Z 896.583,A -85,B 0,C 180,E1 -31684.521,E2 -31684.521} C_VEL
LIN {X 0,Y 128.268,Z 900.289,A -85,B 0,C 180,E1 -31685.29,E2 -31685.29} C_VEL
LIN {X 0,Y 109.564,Z 910.435,A -85,B 0,C 180,E1 -31689.732,E2 -31689.732} C_VEL
LIN {X 0,Y 90.674,Z 919.211,A -85,B 0,C 180,E1 -31696.389,E2 -31696.389} C_VEL
LIN {X 0,Y 73.601,Z 926.094,A -85,B 0,C 180,E1 -31706.282,E2 -31706.282} C_VEL
LIN {X 0,Y 59.253,Z 931.395,A -85,B 0,C 180,E1 -31722.056,E2 -31722.056} C_VEL
LIN {X 0,Y 51.274,Z 934.831,A -85,B 0,C 180,E1 -31744.596,E2 -31744.596} C_VEL
LIN {X 0,Y 51.273,Z 936.254,A -85,B 0,C 180,E1 -31766.647,E2 -31766.647} C_VEL
LIN {X 0,Y 51.777,Z 936.358,A -85,B 0,C 180,E1 -31771.107,E2 -31771.107} C_VEL
LIN {X 0,Y 51.37,Z 935.197,A -85,B 0,C 180,E1 -31791.706,E2 -31791.706} C_VEL
LIN {X 0,Y 58.632,Z 932.116,A -85,B 0,C 180,E1 -31814.364,E2 -31814.364} C_VEL
LIN {X 0,Y 66.259,Z 929.376,A -85,B 0,C 180,E1 -31824.719,E2 -31824.719} C_VEL
LIN {X 0,Y 58.202,Z 922.188,A -85,B 0,C 180,E1 -31873.917,E2 -31873.917} C_VEL
LIN {X 0,Y 74.346,Z 917.75,A -85,B 0,C 180,E1 -31899.777,E2 -31899.777} C_VEL
LIN {X 0,Y 61.243,Z 921.207,A -85,B 0,C 180,E1 -31915.149,E2 -31915.149} C_VEL
LIN {X 0,Y 53.814,Z 922.891,A -85,B 0,C 180,E1 -31934.922,E2 -31934.922} C_VEL
LIN {X 0,Y 52.524,Z 923.167,A -85,B 0,C 180,E1 -31955.461,E2 -31955.461} C_VEL
LIN {X 0,Y 56.954,Z 922.221,A -85,B 0,C 180,E1 -31976.033,E2 -31976.033} C_VEL
LIN {X 0,Y 67.168,Z 919.768,A -85,B 0,C 180,E1 -31993.217,E2 -31993.217} C_VEL
LIN {X 0,Y 81.303,Z 915.72,A -85,B 0,C 180,E1 -32005.485,E2 -32005.485} C_VEL
LIN {X 0,Y 97.815,Z 909.974,A -85,B 0,C 180,E1 -32014.1,E2 -32014.1} C_VEL
LIN {X 0,Y 114.89,Z 902.803,A -85,B 0,C 180,E1 -32020.039,E2 -32020.039} C_VEL
LIN {X 0,Y 132.802,Z 893.809,A -85,B 0,C 180,E1 -32024.521,E2 -32024.521} C_VEL
LIN {X 0,Y 150.347,Z 883.363,A -85,B 0,C 180,E1 -32027.858,E2 -32027.858} C_VEL
LIN {X 0,Y 167.306,Z 871.497,A -85,B 0,C 180,E1 -32030.438,E2 -32030.438} C_VEL
LIN {X 0,Y 183.552,Z 858.193,A -85,B 0,C 180,E1 -32032.495,E2 -32032.495} C_VEL
LIN {X 0,Y 199.003,Z 843.417,A -85,B 0,C 180,E1 -32034.183,E2 -32034.183} C_VEL
LIN {X 0,Y 213.118,Z 827.652,A -85,B 0,C 180,E1 -32035.551,E2 -32035.551} C_VEL
LIN {X 0,Y 214.341,Z 826.119,A -85,B 0,C 180,E1 -32035.683,E2 -32035.683} C_VEL
LIN {X 0,Y 200.329,Z 842.5,A -85,B 0,C 180,E1 -32036.607,E2 -32036.607} C_VEL
LIN {X 0,Y 184.104,Z 858.875,A -85,B 0,C 180,E1 -32037.893,E2 -32037.893} C_VEL
LIN {X 0,Y 166.986,Z 873.731,A -85,B 0,C 180,E1 -32039.585,E2 -32039.585} C_VEL
LIN {X 0,Y 149.058,Z 887.109,A -85,B 0,C 180,E1 -32041.821,E2 -32041.821} C_VEL
LIN {X 0,Y 130.456,Z 899.041,A -85,B 0,C 180,E1 -32044.869,E2 -32044.869} C_VEL
LIN {X 0,Y 128.268,Z 900.289,A -85,B 0,C 180,E1 -32045.29,E2 -32045.29} C_VEL
LIN {X 0,Y 121.603,Z 903.922,A -85,B 0,C 180,E1 -32046.172,E2 -32046.172} C_VEL
LIN {X 0,Y 103.275,Z 912.023,A -85,B 0,C 180,E1 -32047.225,E2 -32047.225} C_VEL
LIN {X 0,Y 96.47,Z 914.829,A -85,B 0,C 180,E1 -32048.532,E2 -32048.532} C_VEL
LIN {X 0,Y 77.923,Z 922.281,A -85,B 0,C 180,E1 -32055.766,E2 -32055.766} C_VEL
LIN {X 0,Y 60.871,Z 928.153,A -85,B 0,C 180,E1 -32067.499,E2 -32067.499} C_VEL
LIN {X 0,Y 47.464,Z 932.458,A -85,B 0,C 180,E1 -32087.615,E2 -32087.615} C_VEL
LIN {X 0,Y 42.535,Z 934.818,A -85,B 0,C 180,E1 -32115.015,E2 -32115.015} C_VEL
LIN {X 0,Y 43.7,Z 935.34,A -85,B 0,C 180,E1 -32131.312,E2 -32131.312} C_VEL
LIN {X 0,Y 44.07,Z 934.072,A -85,B 0,C 180,E1 -32156.987,E2 -32156.987} C_VEL
LIN {X 0,Y 53.64,Z 930.879,A -85,B 0,C 180,E1 -32181.529,E2 -32181.529} C_VEL
LIN {X 0,Y 56.409,Z 929.95,A -85,B 0,C 180,E1 -32185.443,E2 -32185.443} C_VEL
LIN {X 0,Y 50.61,Z 923.709,A -85,B 0,C 180,E1 -32236.057,E2 -32236.057} C_VEL
LIN {X 0,Y 63.763,Z 920.223,A -85,B 0,C 180,E1 -32259.596,E2 -32259.596} C_VEL
LIN {X 0,Y 50.833,Z 923.026,A -85,B 0,C 180,E1 -32277.92,E2 -32277.92} C_VEL
LIN {X 0,Y 44.736,Z 924.146,A -85,B 0,C 180,E1 -32302.292,E2 -32302.292} C_VEL
LIN {X 0,Y 45.931,Z 923.965,A -85,B 0,C 180,E1 -32326.439,E2 -32326.439} C_VEL
LIN {X 0,Y 53.773,Z 922.515,A -85,B 0,C 180,E1 -32347.851,E2 -32347.851} C_VEL
LIN {X 0,Y 67.893,Z 919.273,A -85,B 0,C 180,E1 -32364.097,E2 -32364.097} C_VEL
LIN {X 0,Y 84.388,Z 914.524,A -85,B 0,C 180,E1 -32374.223,E2 -32374.223} C_VEL
LIN {X 0,Y 102.515,Z 908.022,A -85,B 0,C 180,E1 -32381.102,E2 -32381.102} C_VEL
LIN {X 0,Y 121.59,Z 899.619,A -85,B 0,C 180,E1 -32386.016,E2 -32386.016} C_VEL
LIN {X 0,Y 140.319,Z 889.642,A -85,B 0,C 180,E1 -32389.535,E2 -32389.535} C_VEL
LIN {X 0,Y 157.494,Z 878.775,A -85,B 0,C 180,E1 -32392.055,E2 -32392.055} C_VEL
LIN {X 0,Y 174.207,Z 866.376,A -85,B 0,C 180,E1 -32394.07,E2 -32394.07} C_VEL
LIN {X 0,Y 185.336,Z 857.005,A -85,B 0,C 180,E1 -32395.251,E2 -32395.251} C_VEL
LIN {X 0,Y 168.273,Z 871.741,A -85,B 0,C 180,E1 -32396.626,E2 -32396.626} C_VEL
LIN {X 0,Y 149.964,Z 885.325,A -85,B 0,C 180,E1 -32398.472,E2 -32398.472} C_VEL
LIN {X 0,Y 131.006,Z 897.344,A -85,B 0,C 180,E1 -32401.013,E2 -32401.013} C_VEL
LIN {X 0,Y 111.356,Z 907.927,A -85,B 0,C 180,E1 -32404.665,E2 -32404.665} C_VEL
LIN {X 0,Y 96.47,Z 914.829,A -85,B 0,C 180,E1 -32408.532,E2 -32408.532} C_VEL
LIN {X 0,Y 89.644,Z 917.591,A -85,B 0,C 180,E1 -32410.059,E2 -32410.059} C_VEL
LIN {X 0,Y 70.222,Z 923.445,A -85,B 0,C 180,E1 -32413.049,E2 -32413.049} C_VEL
LIN {X 0,Y 63.903,Z 925.186,A -85,B 0,C 180,E1 -32415.641,E2 -32415.641} C_VEL
LIN {X 0,Y 46.757,Z 930.031,A -85,B 0,C 180,E1 -32431.198,E2 -32431.198} C_VEL
LIN {X 0,Y 36.035,Z 933.05,A -85,B 0,C 180,E1 -32458.184,E2 -32458.184} C_VEL
LIN {X 0,Y 35.58,Z 934.334,A -85,B 0,C 180,E1 -32490.001,E2 -32490.001} C_VEL
LIN {X 0,Y 35.468,Z 933.562,A -85,B 0,C 180,E1 -32513.247,E2 -32513.247} C_VEL
LIN {X 0,Y 44.853,Z 930.844,A -85,B 0,C 180,E1 -32543.375,E2 -32543.375} C_VEL
LIN {X 0,Y 46.757,Z 930.33,A -85,B 0,C 180,E1 -32546.514,E2 -32546.514} C_VEL
LIN {X 0,Y 47.552,Z 923.711,A -85,B 0,C 180,E1 -32610.309,E2 -32610.309} C_VEL
LIN {X 0,Y 53.146,Z 922.474,A -85,B 0,C 180,E1 -32619.273,E2 -32619.273} C_VEL
LIN {X 0,Y 40.493,Z 924.644,A -85,B 0,C 180,E1 -32642.019,E2 -32642.019} C_VEL
LIN {X 0,Y 36.479,Z 925.25,A -85,B 0,C 180,E1 -32669.999,E2 -32669.999} C_VEL
LIN {X 0,Y 40.889,Z 924.615,A -85,B 0,C 180,E1 -32699.278,E2 -32699.278} C_VEL
LIN {X 0,Y 53.712,Z 922.421,A -85,B 0,C 180,E1 -32721.43,E2 -32721.43} C_VEL
LIN {X 0,Y 70.909,Z 918.501,A -85,B 0,C 180,E1 -32734.483,E2 -32734.483} C_VEL
LIN {X 0,Y 90.155,Z 912.706,A -85,B 0,C 180,E1 -32742.515,E2 -32742.515} C_VEL
LIN {X 0,Y 109.524,Z 905.326,A -85,B 0,C 180,E1 -32747.645,E2 -32747.645} C_VEL
LIN {X 0,Y 128.501,Z 896.448,A -85,B 0,C 180,E1 -32751.191,E2 -32751.191} C_VEL
LIN {X 0,Y 146.846,Z 886.123,A -85,B 0,C 180,E1 -32753.789,E2 -32753.789} C_VEL
LIN {X 0,Y 155.279,Z 880.743,A -85,B 0,C 180,E1 -32754.828,E2 -32754.828} C_VEL
LIN {X 0,Y 136.207,Z 893.162,A -85,B 0,C 180,E1 -32756.724,E2 -32756.724} C_VEL
LIN {X 0,Y 116.995,Z 903.787,A -85,B 0,C 180,E1 -32759.301,E2 -32759.301} C_VEL
LIN {X 0,Y 97.136,Z 913.051,A -85,B 0,C 180,E1 -32763.155,E2 -32763.155} C_VEL
LIN {X 0,Y 77.931,Z 920.515,A -85,B 0,C 180,E1 -32768.909,E2 -32768.909} C_VEL
LIN {X 0,Y 63.903,Z 925.186,A -85,B 0,C 180,E1 -32775.641,E2 -32775.641} C_VEL
LIN {X 0,Y 57.212,Z 926.945,A -85,B 0,C 180,E1 -32779.022,E2 -32779.022} C_VEL
LIN {X 0,Y 37.624,Z 930.341,A -85,B 0,C 180,E1 -32790.144,E2 -32790.144} C_VEL
LIN {X 0,Y 33.295,Z 931.079,A -85,B 0,C 180,E1 -32797.036,E2 -32797.036} C_VEL
LIN {X 0,Y 26.655,Z 933.023,A -85,B 0,C 180,E1 -32837.249,E2 -32837.249} C_VEL
LIN {X 0,Y 27.496,Z 933.296,A -85,B 0,C 180,E1 -32852.085,E2 -32852.085} C_VEL
LIN {X 0,Y 30.82,Z 931.894,A -85,B 0,C 180,E1 -32892.947,E2 -32892.947} C_VEL
LIN {X 0,Y 36.864,Z 930.547,A -85,B 0,C 180,E1 -32907.977,E2 -32907.977} C_VEL
LIN {X 0,Y 40.901,Z 924.79,A -85,B 0,C 180,E1 -32975.925,E2 -32975.925} C_VEL
LIN {X 0,Y 42.363,Z 924.48,A -85,B 0,C 180,E1 -32978.839,E2 -32978.839} C_VEL
LIN {X 0,Y 30.673,Z 926,A -85,B 0,C 180,E1 -33006.971,E2 -33006.971} C_VEL
LIN {X 0,Y 29.071,Z 926.155,A -85,B 0,C 180,E1 -33041.908,E2 -33041.908} C_VEL
LIN {X 0,Y 38.261,Z 925.075,A -85,B 0,C 180,E1 -33074.877,E2 -33074.877} C_VEL
LIN {X 0,Y 54.841,Z 922.342,A -85,B 0,C 180,E1 -33093.302,E2 -33093.302} C_VEL
LIN {X 0,Y 73.265,Z 918.099,A -85,B 0,C 180,E1 -33102.809,E2 -33102.809} C_VEL
LIN {X 0,Y 92.803,Z 912.143,A -85,B 0,C 180,E1 -33108.654,E2 -33108.654} C_VEL
LIN {X 0,Y 111.959,Z 904.75,A -85,B 0,C 180,E1 -33112.446,E2 -33112.446} C_VEL
LIN {X 0,Y 124.586,Z 899.014,A -85,B 0,C 180,E1 -33114.375,E2 -33114.375} C_VEL
LIN {X 0,Y 104.131,Z 908.971,A -85,B 0,C 180,E1 -33116.993,E2 -33116.993} C_VEL
LIN {X 0,Y 83.006,Z 917.424,A -85,B 0,C 180,E1 -33121.113,E2 -33121.113} C_VEL
LIN {X 0,Y 61.652,Z 924.238,A -85,B 0,C 180,E1 -33128.384,E2 -33128.384} C_VEL
LIN {X 0,Y 42.631,Z 929.047,A -85,B 0,C 180,E1 -33142.041,E2 -33142.041} C_VEL
LIN {X 0,Y 33.295,Z 931.079,A -85,B 0,C 180,E1 -33157.036,E2 -33157.036} C_VEL
LIN {X 0,Y 28.594,Z 931.891,A -85,B 0,C 180,E1 -33168.544,E2 -33168.544} C_VEL
LIN {X 0,Y 23.209,Z 932.353,A -85,B 0,C 180,E1 -33186.054,E2 -33186.054} C_VEL
LIN {X 0,Y 19.156,Z 932.181,A -85,B 0,C 180,E1 -33220.446,E2 -33220.446} C_VEL
LIN {X 0,Y 19.639,Z 931.882,A -85,B 0,C 180,E1 -33237.308,E2 -33237.308} C_VEL
LIN {X 0,Y 27.205,Z 930.505,A -85,B 0,C 180,E1 -33270.273,E2 -33270.273} C_VEL
LIN {X 0,Y 31.561,Z 926.226,A -85,B 0,C 180,E1 -33337.873,E2 -33337.873} C_VEL
LIN {X 0,Y 21.138,Z 927.166,A -85,B 0,C 180,E1 -33376.317,E2 -33376.317} C_VEL
LIN {X 0,Y 24.542,Z 926.922,A -85,B 0,C 180,E1 -33424.775,E2 -33424.775} C_VEL
LIN {X 0,Y 39.509,Z 925.295,A -85,B 0,C 180,E1 -33452.346,E2 -33452.346} C_VEL
LIN {X 0,Y 59.082,Z 921.939,A -85,B 0,C 180,E1 -33464.718,E2 -33464.718} C_VEL
LIN {X 0,Y 79.935,Z 916.787,A -85,B 0,C 180,E1 -33471.183,E2 -33471.183} C_VEL
LIN {X 0,Y 92.966,Z 912.745,A -85,B 0,C 180,E1 -33473.826,E2 -33473.826} C_VEL
LIN {X 0,Y 71.692,Z 920.09,A -85,B 0,C 180,E1 -33477.602,E2 -33477.602} C_VEL
LIN {X 0,Y 50.803,Z 925.709,A -85,B 0,C 180,E1 -33484.515,E2 -33484.515} C_VEL
LIN {X 0,Y 30.931,Z 929.713,A -85,B 0,C 180,E1 -33500.83,E2 -33500.83} C_VEL
LIN {X 0,Y 18.967,Z 931.874,A -85,B 0,C 180,E1 -33545.058,E2 -33545.058} C_VEL
LIN {X 0,Y 19.38,Z 932.272,A -85,B 0,C 180,E1 -33572.959,E2 -33572.959} C_VEL
LIN {X 0,Y 19.639,Z 931.882,A -85,B 0,C 180,E1 -33597.308,E2 -33597.308} C_VEL
LIN {X 0,Y 19.714,Z 931.575,A -85,B 0,C 180,E1 -33607.608,E2 -33607.608} C_VEL
LIN {X 0,Y 18.764,Z 931.02,A -85,B 0,C 180,E1 -33620.395,E2 -33620.395} C_VEL
LIN {X 0,Y 17.044,Z 930.146,A -85,B 0,C 180,E1 -33639.782,E2 -33639.782} C_VEL
LIN {X 0,Y 17.297,Z 928.661,A -85,B 0,C 180,E1 -33677.198,E2 -33677.198} C_VEL
LIN {X 0,Y 20.588,Z 927.773,A -85,B 0,C 180,E1 -33695.862,E2 -33695.862} C_VEL
LIN {X 0,Y 12.802,Z 928.225,A -85,B 0,C 180,E1 -33758.984,E2 -33758.984} C_VEL
LIN {X 0,Y 24.887,Z 927.513,A -85,B 0,C 180,E1 -33812.113,E2 -33812.113} C_VEL
LIN {X 0,Y 44.97,Z 925.165,A -85,B 0,C 180,E1 -33828.047,E2 -33828.047} C_VEL
LIN {X 0,Y 59.429,Z 922.576,A -85,B 0,C 180,E1 -33833.052,E2 -33833.052} C_VEL
LIN {X 0,Y 36.995,Z 927.349,A -85,B 0,C 180,E1 -33840.081,E2 -33840.081} C_VEL
LIN {X 0,Y 16.518,Z 930.278,A -85,B 0,C 180,E1 -33864.778,E2 -33864.778} C_VEL
LIN {X 0,Y 11.259,Z 931.246,A -85,B 0,C 180,E1 -33935.098,E2 -33935.098} C_VEL
LIN {X 0,Y 17.518,Z 930.258,A -85,B 0,C 180,E1 -33995.548,E2 -33995.548} C_VEL
LIN {X 0,Y 17.297,Z 928.661,A -85,B 0,C 180,E1 -34037.198,E2 -34037.198} C_VEL
LIN {X 0,Y 16.915,Z 928.497,A -85,B 0,C 180,E1 -34044.235,E2 -34044.235} C_VEL
LIN {X 0,Y 14.905,Z 928.517,A -85,B 0,C 180,E1 -34052.717,E2 -34052.717} C_VEL
LIN {X 0,Y 10.986,Z 928.707,A -85,B 0,C 180,E1 -34066.171,E2 -34066.171} C_VEL
LIN {X 0,Y 7.287,Z 929.158,A -85,B 0,C 180,E1 -34159.551,E2 -34159.551} C_VEL
LIN {X 0,Y 8.756,Z 929.136,A -85,B 0,C 180,E1 -34168.497,E2 -34168.497} C_VEL
LIN {X 0,Y 22.52,Z 928.504,A -85,B 0,C 180,E1 -34190.777,E2 -34190.777} C_VEL
LIN {X 0,Y 2.818,Z 930.171,A -85,B 0,C 180,E1 -34269.232,E2 -34269.232} C_VEL
LIN {X 0,Y 3.226,Z 930.206,A -85,B 0,C 180,E1 -34311.576,E2 -34311.576} C_VEL
LIN {X 0,Y 8.299,Z 929.821,A -85,B 0,C 180,E1 -34373.081,E2 -34373.081} C_VEL
LIN {X 0,Y 9.592,Z 929.116,A -85,B 0,C 180,E1 -34408.344,E2 -34408.344} C_VEL
LIN {X 0,Y 8.756,Z 929.136,A -85,B 0,C 180,E1 -34528.497,E2 -34528.497} C_VEL
LIN {X 0,Y 10.507,Z 931.136,A -85,B 0,C 180,E1 -34534.617,E2 -34534.617} C_VEL
LIN {X 0,Y 10.507,Z 1012.5,A -85,B 0,C 180,E1 -34534.617,E2 -34534.617} C_VEL
LIN {X 0,Y 10.507,Z 1012.5,A -85,B 0,C 180,E1 -34534.617,E2 -34534.617}

QRS_NEXT_CUT()

QRS_NEXT()
QRS_HOME()

END
